// TIA Portal V16 export
// export: Created 2022-09-01T13:37:04.7970179Z, ExportSetting WithDefaults, DisplayName Totally Integrated Automation Portal, DisplayVersion V16, DisplayName TIA Portal Version Control Interface, DisplayVersion V16, DisplayName TIA Portal Openness, DisplayVersion V16, DisplayName STEP 7 Professional, DisplayVersion V16, DisplayName STEP 7 Safety, DisplayVersion V16, DisplayName WinCC Advanced, DisplayVersion V16
DATA_BLOCK "Inputs_HMI"   // DB14
{ S7_Optimized_Access := 'TRUE' }
VERSION : 0.1
// stored: AutoNumber true, IsOnlyStoredInLoadMemory false, IsRetainMemResEnabled false, IsWriteProtectedInAS false, MemoryReserve 100
   VAR RETAIN
      MODO_1 : Bool;
      MODO_2 : Bool;
   END_VAR
   VAR
      RESET_ALARME : Bool;
      START_CICLO : Bool;
   END_VAR
   VAR RETAIN
      MAN_AUTO : Bool;
   END_VAR
   VAR
      ON_OFF_MX201 : Bool;
      ON_OFF_MX301 : Bool;
      ON_OFF_MX601 : Bool;
      ON_OFF_MX603 : Bool;
      ON_OFF_MX604 : Bool;
      ON_OFF_MX605 : Bool;
      ON_OFF_BD601 : Bool;
      ON_OFF_BD602 : Bool;
      ON_OFF_BD603 : Bool;
      ON_OFF_BD604 : Bool;
      ON_OFF_BD605 : Bool;
      ON_OFF_BS001A : Bool;
      ON_OFF_BS001B : Bool;
      ON_OFF_BS501 : Bool;
      ON_OFF_BH201 : Bool;
      ON_OFF_BM401 : Bool;
      ON_OFF_XV101 : Bool;
      ON_OFF_XV102 : Bool;
   END_VAR
   VAR RETAIN
      TEMP_AREJAMENTO : Time := T#0m;
      TEMP_REDUÇÃO : Time := T#0m;
      TEMP_PRECIPITAÇÃO : Time := T#0m;
      TEMP_ALARME : Time := T#0m;
      TEMP_DOS_COAG : Time;
      HISTERESE : Time;
      SETPOINT_PC401 : Real;
      SP_LSH_TK02 : Real;
      SP_LSM_TK02 : Real;
      SP_LSL_TK02 : Real;
      SP_LSH_TK03 : Real;
      SP_LSM_TK03 : Real;
      SP_LSL_TK03 : Real;
   END_VAR
   VAR
      SALTAR_HISTERESE : Bool;
      RESET_CONT_CICLOS : Bool;
   END_VAR
   VAR RETAIN
      ENABLE_DISABLE_BD603 : Bool := true;
      SUSPENSÃO_CICLO_PRENSA : Bool;
      IGNORAR_LSH101_LSH501 : Bool;
   END_VAR
BEGIN
END_DATA_BLOCK
